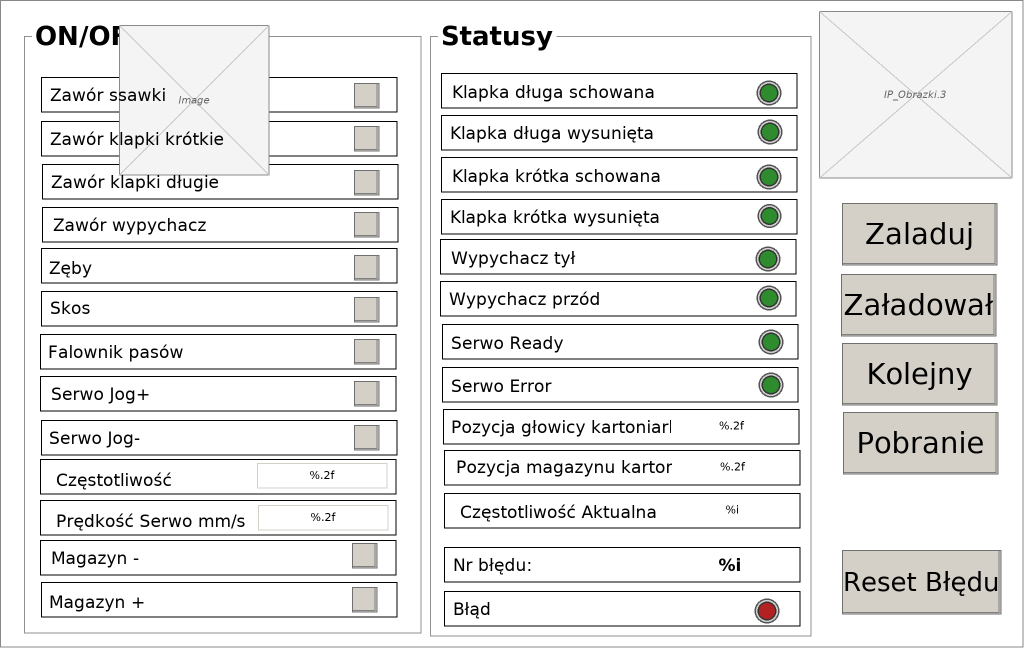
VISUALIZATION Kartoniarka  // 1024x648
    Rectangle (41,121 356x35)
    Rectangle (42,164 356x35)
    Rectangle (42,207 356x35)
    Rectangle (40,334 356x35)
    Rectangle (41,77 356x35)
    Rectangle (41,420 356x35)
    Rectangle (40,376 356x35)
    Rectangle (443,409 356x35)
    GroupBox (430,28 381x608), "Statusy"
        Rectangle (11,129 356x35)
        Rectangle (10,211 356x35)
        Label (18,384 330x30), "Pozycja głowicy kartoniarki"
        Rectangle (14,422 356x35)
        Label (23,424 330x30), "Pozycja magazynu kartonów"
    GroupBox (24,28 397x605), "ON/OFF"
        Rectangle (16,431 356x35)
        Rectangle (16,472 356x35)
        Textfield (234,477 130x25), "%.2f", text variable: gvl_hmi.J_VelK
            OnMouseClick: write the text variable via Edit
        Textfield (233,435 130x25), "%.2f", text variable: GVL_HMI.iFreqKartoniarkaMan
            OnMouseClick: write the text variable via Edit
        Button (330,397 25x25)
            tap GVL_HMI.bHmiJogKF
        Rectangle (17,554 356x35)
        Button (330,55 25x25), colour toggle: GVL_GLOBAL.zaw_ssawki_cewka
            tap GVL_HMI.przycisk_zaw_ssawki
        Button (330,311 25x25), colour toggle: GVL_GLOBAL.falownik_pasow_cewka
            tap GVL_HMI.przycisk_falownik_pasow
        Button (330,184 25x25), colour toggle: GVL_GLOBAL.zaw_wypychacz_cewka
            tap GVL_HMI.przycisk_zaw_wypychacz
        Button (330,142 25x25), colour toggle: GVL_GLOBAL.zaw_klap_dlug_cewka
            tap GVL_HMI.przycisk_zaw_klap_dlug
        Button (330,98 25x25), colour toggle: GVL_GLOBAL.zaw_klap_krot_cewka
            tap GVL_HMI.przycisk_zaw_klap_krot
        Rectangle (17,220 356x35)
        Rectangle (17,263 356x35)
        Label (23,265 209x30), "Skos"
        Button (330,269 25x25), colour toggle: GVL_GLOBAL.zaw_skos_cewka
            tap GVL_HMI.przycisk_zaw_skos
        Button (330,227 25x25), colour toggle: GVL_GLOBAL.zaw_zeby_cewka
            tap GVL_HMI.przycisk_zaw_zeby
        Button (330,353 25x25)
            tap GVL_HMI.bHmiJogKB
        Button (328,559 25x25)
            tap GVL_HMI.bHmiMagCcw
    Image (819,11 193x167), image: IP_Obrazki.3
    Button (842,343 155x62), "Kolejny"
        tap GVL_HMI.Nastepny_Karton
    Image (119,25 150x150)
    Rectangle (441,73 356x35)
    Label (447,76 230x30)
    Rectangle (441,115 356x35)
    Label (447,118 239x30), "Klapka długa wysunięta"
    Lamp1 (756,118 28x28), variable: GVL_IO.Kl_2_wyp, style: Lamp-Lamp1-Green
    Lamp1 (755,79 28x28), variable: GVL_IO.Kl_2_cof, style: Lamp-Lamp1-Green
    Label (449,77 239x30), "Klapka długa schowana"
    Rectangle (442,324 356x35)
    Rectangle (442,367 356x35)
    Label (48,167 209x30), "Zawór klapki długie"
    Label (47,119 239x30)
    Label (47,124 209x30), "Zawór klapki krótkie"
    Label (47,80 209x30), "Zawór ssawki"
    Label (50,210 209x30), "Zawór wypychacz"
    Label (45,337 209x30), "Falownik pasów"
    Label (53,465 209x30), "Częstotliwość"
    Label (448,328 239x30), "Serwo Ready"
    Lamp1 (757,328 28x28), variable: PRG_Kartoniarka.S_Power.Status, style: Lamp-Lamp1-Green
    Label (448,371 239x30), "Serwo Error"
    Lamp1 (757,371 28x28), variable: PRG_Kartoniarka.S_Power.Error, style: Lamp-Lamp1-Green
    Textfield (671,411 121x30), "%.2f", text variable: GVL_AXIS.stAxis1.NcToPlc.ActPos
    Label (48,379 209x30), "Serwo Jog+"
    Label (46,423 209x30), "Serwo Jog-"
    Label (447,160 230x30)
    Rectangle (441,199 356x35)
    Label (447,202 239x30), "Klapka krótka wysunięta"
    Lamp1 (756,202 27x28), variable: GVL_IO.Kl_1_wyp, style: Lamp-Lamp1-Green
    Lamp1 (755,163 28x28), variable: GVL_IO.Kl_1_cof, style: Lamp-Lamp1-Green
    Label (449,161 239x30), "Klapka krótka schowana"
    Label (446,242 230x30)
    Rectangle (440,281 356x35)
    Label (446,284 239x30), "Wypychacz przód"
    Lamp1 (755,284 28x28), variable: GVL_IO.Wyp_wys, style: Lamp-Lamp1-Green
    Lamp1 (754,245 28x28), variable: GVL_IO.Wyp_cof, style: Lamp-Lamp1-Green
    Label (448,243 239x30), "Wypychacz tył"
    Rectangle (444,493 356x35)
    Label (457,497 209x30), "Częstotliwość Aktualna"
    Textfield (672,495 121x30), "%i", text variable: GVL_HMI.iWydajnosc
    Textfield (672,452 121x30), "%.2f", text variable: GVL_AXIS.EC_Magazyn.NcToPlc.ActPos
    Label (53,506 209x30), "Prędkość Serwo mm/s"
    Rectangle (40,540 356x35)
    Button (352,543 25x25)
        tap GVL_HMI.bHmiMagCw
    Label (48,543 209x30), "Magazyn -"
    Label (46,587 209x30), "Magazyn +"
    Button (842,203 155x62), "Zaladuj"
        tap GVL_HMI.zaladuj
    Button (841,274 155x62), "Załadował"
        tap GVL_HMI.zaladowalem
    Button (843,412 155x62), "Pobranie"
        tap GVL_GLOBAL.Zabierz_Z_Kierownicy
    Label (46,253 209x30), "Zęby"
    Rectangle (444,547 356x35)
    Textfield (672,550 116x30), "%i", text variable: GVL_GLOBAL.Error_numb_kart
    Label (450,550 209x30), "Nr błędu:"
    Rectangle (444,591 356x35)
    Label (450,594 209x30), "Błąd"
    Button (842,550 159x64), "Reset Błędu"
        tap GVL_GLOBAL.Error_reset_kart
    Lamp1 (753,597 28x28), variable: GVL_GLOBAL.Error_ind_kart, style: Lamp-Lamp1-Red
END_VISUALIZATION

(* stored: Version 1.1.0.1, ProductVersion 3.1.4022.12
   Visu Kartoniarka: Id {fb2af1fe-4f36-4274-ab2a-e62d0a11dee0} *)
